# B&R Automation Studio project Nitto (part 9)

### RCP_glob.var - Package variables
```iecst
(********************************************************************
 * COPYRIGHT -- Bernecker + Rainer
 ********************************************************************
 * File: RCP_glob.var
 * Author: beutert
 * Created: September 07, 2012
 ********************************************************************
 * Global variables of project csv_bsp
 ********************************************************************)
(*======================================================================================================================================*)
(*Global recipe constants*)
(*======================================================================================================================================*)
VAR CONSTANT
	RCP_PROG_TEXT_DESCRIPTION_MAX : UINT := 79; (*maximale Anzahl von Zeichen für Beschreibungen für Rezept und Zeile*)
	RCP_PROG_TEXT_FILENAME_MAX : UINT := 29; (*maximale Anzahl von Zeichen für den Rezeptnamen*)
END_VAR
(*======================================================================================================================================*)
(*Global recipe variables*)
(*======================================================================================================================================*)
VAR
	Button : Button_typ := (0);
	ToolEdit : rcp_tool_typ := (0);
	RecipeEdit : rcp_prog_typ := (0);
	RecipeWork : rcp_prog_typ := (0);
END_VAR
```

### Glob_IO.typ - Package data types
```iecst
(********************************************************************
 * COPYRIGHT -- Bernecker + Rainer
 ********************************************************************
 * File: Glob_IO.typ
 * Author: schoenefeldr
 * Created: July 10, 2012
 ********************************************************************
 * Global data types of project 120706_hp_001
 ********************************************************************)

TYPE
	MachineIoDi_Type : 	STRUCT
		FuseFanUnwind : DiDo_Type; (*Sicherung Lüfter Abwicklung*)
		FusePlug1 : DiDo_Type; (*Sicherung OK Schukosteckdose 1*)
		FusePlug2 : DiDo_Type; (*Sicherung OK Schukosteckdose 2*)
		FusePlugCEE : DiDo_Type; (*Sicherung OK CEE-Steckdose*)
		FuseBTS : DiDo_Type; (*Sicherung OK Bahnkantensteuerung*)
		FuseQW258_262 : DiDo_Type; (*Sicherung OK QW258 - QW262*)
		FuseQW264_268 : DiDo_Type; (*Sicherung OK QW264 - QW268*)
		FuseBookletFeeder : DiDo_Type; (*Sicherung OK Booklet Feeder*)
		FuseHydraulicPump : DiDo_Type; (*Sicherung OK Hydraulikpumpe*)
		HighVoltageGenerator : DiDo_Type; (*Hochspannungsgenerator Anti-Statik OK / Ein-Aus*)
		BST_OK : DiDo_Type; (*BST OK*)
		RFK_EmcyStop_undelayed : DiDo_Type; (*RFK Not - Halt - Schütze unverzögert*)
		RFK_EmcyStop_delayed : DiDo_Type; (*RFK Not - Halt - Schütze verzögert*)
		LDT_Reset : DiDo_Type; (*LDT Reset / Steuerung Ein*)
		LDT_CtrlOff : DiDo_Type; (*LDT Steuerung Aus*)
		LDT_AutoStart_End : DiDo_Type; (*LDT Automatik Start Maschinenende*)
		LDT_AutoStart_Middle : DiDo_Type; (*LDT Automatik Start Maschinenmitte*)
		LDT_AutoStart_Unwind : DiDo_Type; (*LDT Automatik Start am Abwickler*)
		LDT_AutoStart : DiDo_Type; (*LDT Automatik Start*)
		LDT_AutoStop : DiDo_Type; (*LDT Automatik Stopp*)
		LDT_AutoStop_End : DiDo_Type; (*LDT Automatik Stopp Maschinenende*)
		LDT_AutoStop_Middle : DiDo_Type; (*LDT Automatik Stopp Maschinenmitte*)
		LDT_AutoStop_Unwind : DiDo_Type; (*LDT Automatik Stopp am Abwickler*)
		LDT_Reserve2 : DiDo_Type;
		LDT_Jog_Machine : DiDo_Type; (*LDT Jog-Mode*)
		LDT_Jog_Machine_End : DiDo_Type; (*LDT Jog-Mode Maschinenende*)
		LDT_Jog_Machine_Middle : DiDo_Type; (*LDT Jog-Mode Maschinenmitte*)
		LDT_Jog_Machine_Unwind : DiDo_Type; (*LDT Jog-Mode am Abwickler*)
		LDT_Reserve1 : DiDo_Type;
		LDT_FaultReset : DiDo_Type; (*LDT Störung quittieren*)
		LDT_UnwindMoveUp : DiDo_Type; (*LDT Abwickler heben*)
		LDT_Laminator_UpDn : DiDo_Type;
		LDT_LabelDisp_UpDn : DiDo_Type;
		LDT_UnwindMoveDown : DiDo_Type; (*LDT Abwickler senken*)
		LDT_PBS2_upDn : DiDo_Type; (*LDT Zugeinheit heben / senken*)
		LDT_LongCUTsetKnife : DiDo_Type; (*Taster zum Einsetzen der Messer*)
		LDT_PBU_upDn : DiDo_Type; (*LDT Zugstation 3 heben / senken*)
		LDT_CutTabInfeed : DiDo_Type; (*LDT Schneidetisch heben / senken Einlaufseite*)
		LDT_CutTabOutfeed : DiDo_Type; (*LDT Schneidetisch heben / senken Auslaufseite*)
		LDT_PBS1_upDn : DiDo_Type; (*LDT Zugstation 1 heben / senken*)
		LDT_LongCutUpDn : DiDo_Type; (*LDT Längsschneider heben / senken*)
		RD_UnwindTopPos : DiDo_Type; (*RD Abwickler oben*)
		RD_UnwindBotPos : DiDo_Type; (*RD Abwickler unten*)
		RD_PBS1_topPos : DiDo_Type; (*RD Zugstation 1 oben*)
		RD_PBS1_botPos : DiDo_Type; (*RD Zugstation 1 unten*)
		RD_PBU_topPos : DiDo_Type; (*RD Zugstation 3 oben*)
		RD_PBU_botPos : DiDo_Type; (*RD Zugstation 3 unten*)
		Cut1_Ref : DiDo_Type; (*Stanze 1 Referenzpunkt*)
		Cut2_Ref : DiDo_Type; (*Stanze 2 Referenzpunkt*)
		Cut3_Ref : DiDo_Type; (*Stanze 2 Referenzpunkt*)
		RD_PBS2_topPos : DiDo_Type; (*RD Zugeinheit oben*)
		RD_PBS2_botPos : DiDo_Type; (*RD Zugeinheit unten*)
		RD_LongCutTopPos : DiDo_Type; (*RD Längsschneider oben*)
		RD_LongCutBotPos : DiDo_Type; (*RD Längsschneider unten*)
		PressureCtrl : DiDo_Type; (*Druckwächter*)
		SafetyDoorInfeedCut1 : DiDo_Type; (*Safety Door Stanze 1 Infeed*)
		SafetyDoorOutfeedCut1 : DiDo_Type; (*Safety Door Stanze 1 Outfeed*)
		SafetyDoorInfeedCut2 : DiDo_Type; (*Safety Door Stanze 2 Infeed*)
		SafetyDoorOutfeedCut2 : DiDo_Type; (*Safety Door Stanze 2 Outfeed*)
		SafetyDoorInfeedCut3 : DiDo_Type; (*Safety Door Stanze 3 Infeed*)
		SafetyDoorOutfeedCut3 : DiDo_Type; (*Safety Door Stanze 3 Outfeed*)
		SafetyDoorLongCut : DiDo_Type; (*Safety Door Long cut unit*)
		SafetyDoorBooklet : DiDo_Type; (*Safety Door Long cut unit*)
		EmergencyStopCabinet : DiDo_Type; (*Not-Aus-Schalter am Schaltschrank*)
		EmergencyStopPanel : DiDo_Type; (*Not-Aus-Schalter am Panel*)
		EmergencyStopUnwinder : DiDo_Type; (*Not-Aus-Schalter am Abwickler*)
		EmergencyStopBooklet : DiDo_Type; (*Not-Aus-Schalter am Schaltschrank*)
		EmergencyStopLongCut : DiDo_Type; (*Not-Aus-Schalter am Längsschneider*)
		EmergencyStopPullWire : DiDo_Type; (*Not-Aus-Schalter am Längsschneider*)
		LightSensorConvBelt : DiDo_Type; (*Lichttaster Auslageband*)
		EmergencyStopTandemWinder : DiDo_Type; (*Not-Aus-Schalter am Tandemwickler*)
		EmergencyStopEndModule : DiDo_Type; (*Not-Aus-Schalter am Ende der Maschine*)
		EmergencyStopMiddle : DiDo_Type; (*Not-Aus-Schalter in der Mitte der Maschine*)
		RD_LaminatorTopPos : DiDo_Type;
		RD_LaminatorBotPos : DiDo_Type;
		LT_LabelDisp_LoopUnwinder : DiDo_Type;
		LT_LabelDisp_LoopWinder : DiDo_Type;
		LT_LabelDisp_WebBreak1 : DiDo_Type;
		LT_LabelDisp_WebBreak2 : DiDo_Type;
		LabelDisp_RegMark1 : DiDo_Type;
		LabelDisp_RegMark2 : DiDo_Type;
		Fuse_Laminator1 : DiDo_Type;
		Fuse_Laminator2 : DiDo_Type;
		Fuse_GridWinder1 : DiDo_Type;
		Fuse_LabelDisp1 : DiDo_Type;
		Fuse_LabelDisp2 : DiDo_Type;
		TopWindSpikeSuppClosed : DiDo_Type;
		Liner_detekce : DiDo_Type;
		BotWindSpikeSuppClosed : DiDo_Type;
	END_STRUCT;
	MachineIo_Type : 	STRUCT
		DIn : MachineIoDi_Type;
		DOut : MachineIoDo_Type;
		AIn : MachineIoAi_Type;
		AOut : MachineIoAo_Type;
	END_STRUCT;
	MachineIoDo_Type : 	STRUCT
		CtrlPowerEmcyUndel : DiDo_Type; (*24V DC Versorgung nach Not-Halt*)
		CtrlPowerEmcyDel : DiDo_Type; (*24V DC Versorgung nach Not-Halt zeitverzögert*)
		EnabDrives : DiDo_Type; (*Enable ACOPOS-Multi*)
		ContactSuction : DiDo_Type; (*potentialfreier Kontakt Absaugung Ein*)
		Plug1_OnOff : DiDo_Type; (*Schukosteckdose 1 Ein / Aus*)
		Plug2_OnOff : DiDo_Type; (*Schukosteckdose 2 Ein / Aus*)
		PlugCEE_OnOff : DiDo_Type; (*CEE-Steckdose 16A Ein / Aus*)
		HydraulicPumpOn : DiDo_Type; (*Schütz Hydraulikpumpe ein*)
		BST_Enable : DiDo_Type; (*BST Freigabe*)
		BST_Manual : DiDo_Type; (*BST Handbetrieb*)
		BST_Neutral : DiDo_Type; (*BST Mittenstellung*)
		BST_Automatic : DiDo_Type; (*BST Mittenstellung*)
		BST_ArrowLeft : DiDo_Type; (*BST Pfeil links BST Tastatursperre*)
		BST_ArrowRight : DiDo_Type; (*BST Pfeil rechts BST Tastatursperre*)
		LampGreen : DiDo_Type; (*Turmleuchte grün*)
		LampYellow : DiDo_Type; (*Turmleuchte gelb*)
		LampRed : DiDo_Type; (*Turmleuchte rot*)
		TowerHorn : DiDo_Type; (*Turmleuchte Hupe*)
		VentLabelDisp : DiDo_Type; (*Ventil Label Dispenser Up Down*)
		VentLaminatorMoveUp : DiDo_Type; (*Ventil Abwickler heben*)
		VentLaminatorMoveDown : DiDo_Type; (*Ventil Abwickler heben*)
		VentUnwindMoveUp : DiDo_Type; (*Ventil Laminierer heben*)
		VentUnwindMoveDown : DiDo_Type; (*Ventil Laminierer senken*)
		VentCutTabInfeedMoveUpDn : DiDo_Type; (*Ventil Schneidetisch heben / senken Einlaufseite*)
		VentCutTabOutfeedMoveUpDn : DiDo_Type; (*Ventil Schneidetisch heben / senken Auslaufseite*)
		Vent1Dancer : DiDo_Type; (*Ventil 1 Tänzer*)
		VentAirSupply : DiDo_Type; (*Hauptventil*)
		VentPBS1_MoveDown : DiDo_Type; (*Ventil Zugstation 1 senken*)
		VentPBS1_MoveUp : DiDo_Type; (*Ventil Zugstation 1 heben*)
		VentPBU_MoveUP : DiDo_Type; (*Ventil Zugstation 3 heben*)
		VentPBU_MoveDown : DiDo_Type; (*Ventil Zugstation 3 senken*)
		VentPBS2_MoveDown : DiDo_Type; (*Ventil Zugeinheit senken*)
		VentLongCutMoveUp : DiDo_Type; (*Ventil Längsschneider heben*)
		VentLongCutSetKnifeIn : DiDo_Type; (*Ventil Längsschneider Messer setzen*)
		VentLongCutSetKnifeOut : DiDo_Type; (*Ventil Längsschneider Messer setzen*)
		VentLongCutMoveDown : DiDo_Type; (*Ventil Längsschneider senken *)
		ValveCuttingUnitToolUp : DiDo_Type; (*Ventil Stanzstation Werkzeug heben*)
		ValveCut1BridgeDown : DiDo_Type; (*Ventil Stanzstation1 Brücke senken*)
		ValveCut2BridgeDown : DiDo_Type; (*Ventil Stanzstation 2 Brücke senken*)
		ValveCut3BridgeDown : DiDo_Type; (*Ventil Stanzstation 3 Brücke senken*)
		BookletFeederREG : DiDo_Type; (*Ventil Stanzstation 3 Brücke senken*)
		BookletFeederON : DiDo_Type; (*Ventil Stanzstation 3 Brücke senken*)
	END_STRUCT;
	MachineIoAo_Type : 	STRUCT
		MagBrakeUnwind : AiAo_Type; (*Ansteuerung Magnetpulverbremse Abwickler*)
		VentDancer : AiAo_Type; (*Proportionalventil Tänzerspannung (Festo)*)
		VentClutchSpend1 : AiAo_Type; (*Proportionalventil Rutschkupplung Abwickler 1*)
		VentClutchSpend2 : AiAo_Type; (*Proportionalventil Rutschkupplung Abwickler 2*)
		VentClutchSpend3 : AiAo_Type; (*Proportionalventil Rutschkupplung Abwickler 3*)
		VentClutchLaminator1 : AiAo_Type; (*Proportionalventil Rutschkupplung Abwickler 3*)
		VentClutchLaminator2 : AiAo_Type; (*Proportionalventil Rutschkupplung Abwickler 3*)
		VentClutchGrid1 : AiAo_Type; (*Proportionalventil Rutschkupplung Gitteraufwickler 1*)
		VentClutchGrid2 : AiAo_Type; (*Proportionalventil Rutschkupplung Gitteraufwickler 2*)
		VentOptClutchTUnwindTop : AiAo_Type; (*Option Proportionalventil Rutschkupplung Tandemwickler oben*)
		VentOptClutchTUnwindBot : AiAo_Type; (*Option Proportionalventil Rutschkupplung Tandemwickler unten*)
	END_STRUCT;
	MachineIoAi_Type : 	STRUCT
		FlengeDMS : AiAo_Type; (*Flanschkraftaufnehmer*)
		FDriveSideCut1 : AiAo_Type; (*Stanze 1 Druckkraftaufnehmer Antriebsseite*)
		FOperatorSideCut1 : AiAo_Type; (*Stanze 1 Druckkraftaufnehmer Bedienerseite*)
		FDriveSideCut2 : AiAo_Type; (*Stanze 2 Druckkraftaufnehmer Antriebsseite*)
		FOperatorSideCut2 : AiAo_Type; (*Stanze 2 Druckkraftaufnehmer Bedienerseite*)
		FDriveSideCut3 : AiAo_Type; (*Stanze 3 Druckkraftaufnehmer Antriebsseite*)
		FOperatorSideCut3 : AiAo_Type; (*Stanze 3 Druckkraftaufnehmer Bedienerseite*)
		DiamMainUnwind : AiAo_Type; (*Durchmesserabfrage Abwicklung*)
		DiamSpend1 : AiAo_Type; (*Durchmesserabfrage Abwickler 1*)
		DiamSpend2 : AiAo_Type; (*Durchmesserabfrage Abwickler 2*)
		DiamLaminator1 : AiAo_Type; (*Durchmesserabfrage Laminierer 1*)
		DiamLaminator2 : AiAo_Type; (*Durchmesserabfrage Laminierer 2*)
		DiamGrid1 : AiAo_Type; (*Durchmesserabfrage Gitteraufwickler 1*)
		DiamGrid2 : AiAo_Type; (*Durchmesserabfrage Gitteraufwickler 2*)
		DancerPos : AiAo_Type; (*Tänzerlage*)
		DiamTUnwindTop : AiAo_Type; (*Durchmesserabfrage Tandemwickler oben*)
		DiamTUnwindBot : AiAo_Type; (*Durchmesserabfrage Tandemwickler unten*)
		Dancer_position : AiAo_Type; (*pozice danceru optický senzor*)
		TestSensor : AiAo_Type; (*Durchmesserabfrage Tandemwickler unten*)
	END_STRUCT;
END_TYPE
```

### Library Logical/Bibliothek (IEC) - Eine neue Quellbibliothek

#### Package Logical/Bibliothek/CONST - Neues leeres Paket

#### FB_CONST_AXISSTATE.st
```iecst
(********************************************************************
 * COPYRIGHT -- Microsoft
 ********************************************************************
 * Library: Bibliothek
 * Datei: FB_CONST_AXISSTATE.st
 * Autor: awalz
 * Erstellt: 26. August 2014
 ********************************************************************
 * Implementierung der Library Bibliothek
 ********************************************************************)

(* TODO: Bitte Kommentar hier einfügen *)
FUNCTION_BLOCK FB_CONST_AXIS_STATE
END_FUNCTION_BLOCK
```

#### FB_CONST_UNIT_MODES.st
```iecst
(********************************************************************
 * COPYRIGHT -- Microsoft
 ********************************************************************
 * Library: Bibliothek
 * Datei: FB_CONST_UNIT_MODES.st
 * Autor: Awalz
 * Erstellt: 7. Mai 2014
 ********************************************************************
 * Implementierung der Library Bibliothek
 ********************************************************************)

 (*<$Description$> TODO: Bitte Kommentar hier einzufügen </$Description$>*)
FUNCTION_BLOCK FB_CONST_UNIT_MODES
END_FUNCTION_BLOCK
```

#### FB_CONST_CUTTINGUNIT_CMDS.st
```iecst
(********************************************************************
 * COPYRIGHT -- Microsoft
 ********************************************************************
 * Library: Bibliothek
 * Datei: FB_CONST_CUTTINGUNIT_CMDS.st
 * Autor: Awalz
 * Erstellt: 7. Mai 2014
 ********************************************************************
 * Implementierung der Library Bibliothek
 ********************************************************************)

 (*<$Description$> TODO: Bitte Kommentar hier einzufügen </$Description$>*)
FUNCTION_BLOCK FB_CONST_CUTTINGUNIT_CMDS
END_FUNCTION_BLOCK
```

#### FB_CONST_CUTTINGUNIT_MODES.st
```iecst
(********************************************************************
 * COPYRIGHT -- Microsoft
 ********************************************************************
 * Library: Bibliothek
 * Datei: FB_CONST_CUTTINGUNIT_MODES.st
 * Autor: Awalz
 * Erstellt: 7. Mai 2014
 ********************************************************************
 * Implementierung der Library Bibliothek
 ********************************************************************)

 (*<$Description$> TODO: Bitte Kommentar hier einzufügen </$Description$>*)
FUNCTION_BLOCK FB_CONST_CUTTINGUNIT_MODES
END_FUNCTION_BLOCK
```

#### FB_CONST_MASCHINE.st
```iecst
(********************************************************************
 * COPYRIGHT -- Microsoft
 ********************************************************************
 * Library: Bibliothek
 * Datei: FB_CONST_MASCHINE.st
 * Autor: Awalz
 * Erstellt: 1. April 2014
 ********************************************************************
 * Implementierung der Library Bibliothek
 ********************************************************************)

 (*<$Description$> TODO: Bitte Kommentar hier einzufügen </$Description$>*)
FUNCTION_BLOCK FB_CONST_MASCHINE
END_FUNCTION_BLOCK
```

#### FB_CONST_AXIS_ACTIONS.st
```iecst
(********************************************************************
 * COPYRIGHT -- Microsoft
 ********************************************************************
 * Library: Bibliothek
 * Datei: FB_CONST_AXIS_ACTIONS.st
 * Autor: Awalz
 * Erstellt: 1. April 2014
 ********************************************************************
 * Implementierung der Library Bibliothek
 ********************************************************************)

 (*<$Description$> TODO: Bitte Kommentar hier einzufügen </$Description$>*)
FUNCTION_BLOCK FB_CONST_AXIS_ACTIONS
END_FUNCTION_BLOCK
```

#### FB_CONST_MACHINE_MODE.st
```iecst
(********************************************************************
 * COPYRIGHT -- Microsoft
 ********************************************************************
 * Library: Bibliothek
 * Datei: FB_CONST_MACHINE_MODE.st
 * Autor: Awalz
 * Erstellt: 31. März 2014
 ********************************************************************
 * Implementierung der Library Bibliothek
 ********************************************************************)

 (*<$Description$> TODO: Bitte Kommentar hier einzufügen </$Description$>*)
FUNCTION_BLOCK FB_CONST_MACHINE_MODES
END_FUNCTION_BLOCK
```

#### FB_CONST_LAMP.st
```iecst
(********************************************************************
 * COPYRIGHT -- Microsoft
 ********************************************************************
 * Library: Bibliothek
 * Datei: FB_CONST_LAMP.st
 * Autor: Awalz
 * Erstellt: 30. April 2014
 ********************************************************************
 * Implementierung der Library Bibliothek
 ********************************************************************)

 (*<$Description$> TODO: Bitte Kommentar hier einzufügen </$Description$>*)
FUNCTION_BLOCK FB_CONST_LAMP
END_FUNCTION_BLOCK
```

#### FB_CONST_CUTTINGUNIT.st
```iecst
(********************************************************************
 * COPYRIGHT -- Microsoft
 ********************************************************************
 * Library: Bibliothek
 * Datei: FB_CONST_CUTTINGUNIT.st
 * Autor: Awalz
 * Erstellt: 7. Mai 2014
 ********************************************************************
 * Implementierung der Library Bibliothek
 ********************************************************************)

 (*<$Description$> TODO: Bitte Kommentar hier einzufügen </$Description$>*)
FUNCTION_BLOCK FB_CONST_CUTTINGUNIT
END_FUNCTION_BLOCK
```

#### FB_CUTTINGUNIT_CMD.st
```iecst
(********************************************************************
 * COPYRIGHT -- Microsoft
 ********************************************************************
 * Library: Bibliothek
 * Datei: FB_CUTTINGUNIT_CMD.st
 * Autor: Awalz
 * Erstellt: 7. Mai 2014
 ********************************************************************
 * Implementierung der Library Bibliothek
 ********************************************************************)

 (*<$Description$> TODO: Bitte Kommentar hier einzufügen </$Description$>*)
FUNCTION_BLOCK FB_CUTTINGUNIT_CMD
	IF set THEN
		IF value < CONST.CUTTINGUNIT.CMDs.NO_CMD OR value > CONST.CUTTINGUNIT.CMDs.ABORT THEN
			text := '******';
		ELSE
			text := CONST.CUTTINGUNIT.CMDs.texts[value];
		END_IF
	END_IF
END_FUNCTION_BLOCK
```

#### FB_CUTTING_MODE.st
```iecst
(********************************************************************
 * COPYRIGHT -- Microsoft
 ********************************************************************
 * Library: Bibliothek
 * Datei: FB_CUTTING_MODE.st
 * Autor: Awalz
 * Erstellt: 20. Mai 2014
 ********************************************************************
 * Implementierung der Library Bibliothek
 ********************************************************************)

 (*<$Description$> TODO: Bitte Kommentar hier einzufügen </$Description$>*)
FUNCTION_BLOCK FB_CUTTING_MODE
END_FUNCTION_BLOCK
```

#### FB_CONST_CUTTINGUNIT_TOOLS.st
```iecst
(********************************************************************
 * COPYRIGHT -- Microsoft
 ********************************************************************
 * Library: Bibliothek
 * Datei: FB_CONST_CUTTINGUNIT_TOOLS.st
 * Autor: okrebs
 * Erstellt: 23. Mai 2014
 ********************************************************************
 * Implementierung der Library Bibliothek
 ********************************************************************)

(* TODO: Bitte Kommentar hier einzufügen *)
FUNCTION_BLOCK FB_CONST_CUTTINGUNIT_TOOLS
END_FUNCTION_BLOCK
```

#### FB_CONST_ALARMS.st
```iecst
(********************************************************************
 * COPYRIGHT -- Microsoft
 ********************************************************************
 * Library: Bibliothek
 * Datei: FB_CONST_ALARMS.st
 * Autor: awalz
 * Erstellt: 1. August 2014
 ********************************************************************
 * Implementierung der Library Bibliothek
 ********************************************************************)

(* TODO: Bitte Kommentar hier einfügen *)
FUNCTION_BLOCK FB_CONST_ALARMS
END_FUNCTION_BLOCK
```

#### FB_CONST_CUTTINGUNIT_ERRORS.st
```iecst
(********************************************************************
 * COPYRIGHT -- Microsoft
 ********************************************************************
 * Library: Bibliothek
 * Datei: FB_CONST_CUTTINGUNIT_ERRORS.st
 * Autor: okrebs
 * Erstellt: 23. Mai 2014
 ********************************************************************
 * Implementierung der Library Bibliothek
 ********************************************************************)

(* TODO: Bitte Kommentar hier einzufügen *)
FUNCTION_BLOCK FB_CONST_CUTTINGUNIT_ERRORS
END_FUNCTION_BLOCK
```

#### Package Logical/Bibliothek/Genarals - Neues leeres Paket

#### FB_Lamp.st
```iecst
(********************************************************************
 * COPYRIGHT -- Microsoft
 ********************************************************************
 * Library: Bibliothek
 * Datei: FB_Lamp.st
 * Autor: Awalz
 * Erstellt: 12. Mai 2014
 ********************************************************************
 * Implementierung der Library Bibliothek
 ********************************************************************)

 (*<$Description$> TODO: Bitte Kommentar hier einzufügen </$Description$>*)
FUNCTION_BLOCK FB_Lamp
 rtrig(CLK := button);
	ftrig(CLK := button);
 	IF aktion = CONST.LAMP.OFF THEN
 		output := FALSE;
	ELSIF aktion = CONST.LAMP.ON THEN
		output := TRUE;
	ELSIF aktion = CONST.LAMP.BLINK200 THEN
		output := clk.c200.Output;
	ELSIF aktion = CONST.LAMP.BLINK500 THEN
		output := clk.c500.Output;
	ELSIF aktion = CONST.LAMP.BLINK1000 THEN
		output := clk.c1000.Output;
	ELSIF aktion = CONST.LAMP.BLINK5000 THEN
		output := clk.c5000.Output;
	END_IF

	led := output;
	ledinv := NOT output;

END_FUNCTION_BLOCK
```

#### FB_Clk.st
```iecst
(********************************************************************
 * COPYRIGHT -- Microsoft
 ********************************************************************
 * Library: Bibliothek
 * Datei: FB_Clk.st
 * Autor: Awalz
 * Erstellt: 30. April 2014
 ********************************************************************
 * Implementierung der Library Bibliothek
 ********************************************************************)

 (*<$Description$> TODO: Bitte Kommentar hier einzufügen </$Description$>*)
FUNCTION_BLOCK FB_Clk
	c200();
	c500();
	c1000();
	c5000();
END_FUNCTION_BLOCK
```

#### FB_KeyLamp.st
```iecst
(********************************************************************
 * COPYRIGHT -- Microsoft
 ********************************************************************
 * Library: Bibliothek
 * Datei: FB_KeyLamp.st
 * Autor: Awalz
 * Erstellt: 12. Mai 2014
 ********************************************************************
 * Implementierung der Library Bibliothek
 ********************************************************************)

 (*<$Description$> TODO: Bitte Kommentar hier einzufügen </$Description$>*)
FUNCTION_BLOCK FB_KeyLamp
		LDT( clk := clk );
END_FUNCTION_BLOCK
```

#### FB_Ampel.st
```iecst
(********************************************************************
 * COPYRIGHT -- Microsoft
 ********************************************************************
 * Library: Bibliothek
 * Datei: FB_Ampel.st
 * Autor: Awalz
 * Erstellt: 12. Mai 2014
 ********************************************************************
 * Implementierung der Library Bibliothek
 ********************************************************************)

 (*<$Description$> TODO: Bitte Kommentar hier einzufügen </$Description$>*)
FUNCTION_BLOCK FB_Ampel
	rtrig(CLK := horn);
	hornPuls(clk := clk);
	Rot(clk := clk);
	Gelb(clk := clk);
	Gruen(clk := clk);
	timer_TOF(IN := rtrig.Q, PT := ondelay);
//	horn_o := timer_TOF.Q;
	horn_o := SEL (timer_TOF.Q, hornPuls.led, timer_TOF.Q); (* pulsierendes Hupen zu erzeugen das Signal wird durch hornPuls von Aussen getaktet*)
END_FUNCTION_BLOCK
```

#### FB_ModulStatus.st
```iecst
(********************************************************************
 * COPYRIGHT -- Microsoft
 ********************************************************************
 * Library: Bibliothek
 * Datei: FB_ModulStatus.st
 * Autor: Awalz
 * Erstellt: 12. Mai 2014
 ********************************************************************
 * Implementierung der Library Bibliothek
 ********************************************************************)

 (*<$Description$> TODO: Bitte Kommentar hier einzufügen </$Description$>*)
FUNCTION_BLOCK FB_ModulStatus
	IF axisState.ContinuousMotion THEN
		AxisState_status := 'ContinuousMotion';
	ELSIF axisState.Disabled THEN
		AxisState_status := 'Disabled';
	ELSIF axisState.DiscreteMotion THEN
		AxisState_status := 'DiscreteMotion';
	ELSIF axisState.Error THEN
		AxisState_status := 'Error';
	ELSIF axisState.Errorstop THEN
		AxisState_status := 'Errorstop';
	ELSIF axisState.StandStill THEN
		AxisState_status := 'StandStill';
	ELSIF axisState.Stopping THEN
		AxisState_status := 'Stopping';
	ELSIF axisState.SynchronizedMotion THEN
		AxisState_status := 'SynchronizedMotion';
	END_IF
END_FUNCTION_BLOCK
```

#### FB_UnitChkStatus.st
```iecst
(********************************************************************
 * COPYRIGHT -- Microsoft
 ********************************************************************
 * Library: Bibliothek
 * Datei: FB_UnitChkStatus.st
 * Autor: Awalz
 * Erstellt: 12. Mai 2014
 ********************************************************************
 * Implementierung der Library Bibliothek
 ********************************************************************)

 (*<$Description$> TODO: Bitte Kommentar hier einzufügen </$Description$>*)
FUNCTION_BLOCK FB_UnitChkStatus
	IF enable THEN
		IF setMode = status.mode THEN
			IF setMode = CONST.UNITMODEs.DISABLE THEN
				ready := NOT status.isCoupled;
			ELSIF setMode = CONST.UNITMODEs.ENABLE THEN
				ready := status.isCoupled;
			ELSE
				ready := FALSE;
			END_IF
		ELSE
			ready := FALSE;
		END_IF
	END_IF

	status.ready := ready;
END_FUNCTION_BLOCK
```

#### FB_ClkPulse.st
```iecst
(********************************************************************
 * COPYRIGHT -- Microsoft
 ********************************************************************
 * Library: Bibliothek
 * Datei: FB_ClkPulse.st
 * Autor: Awalz
 * Erstellt: 30. April 2014
 ********************************************************************
 * Implementierung der Library Bibliothek
 ********************************************************************)

 (*<$Description$> TODO: Bitte Kommentar hier einzufügen </$Description$>*)
FUNCTION_BLOCK FB_ClkPulse

CASE state OF
	CLOCK_ON:
		IF enable THEN
			Output := TRUE;
			timer(IN := FALSE);
			timer(IN := TRUE, PT := TimeOn);
		  	state:= CLOCK_WAIT_ON;
		END_IF

	CLOCK_WAIT_ON:
		timer();
		IF NOT enable THEN
			timer(IN := FALSE);
			Output := FALSE;
			state := CLOCK_ON;
		ELSIF timer.Q THEN
			timer(IN := FALSE);
			Output := FALSE;
			timer(IN := TRUE, PT := TimeOff);
	   		state := CLOCK_WAIT_OFF;
		END_IF

	CLOCK_WAIT_OFF:
		timer();
		IF NOT enable THEN
			timer(IN := FALSE);
			Output := FALSE;
			state := CLOCK_ON;
		ELSIF timer.Q THEN
			Output := TRUE;
			timer(IN := FALSE);
			timer(IN := TRUE, PT := TimeOn);
		   	state:= CLOCK_WAIT_ON;
		END_IF
	ELSE  						(* Unknown program state *)
		state:= CLOCK_ON;
	END_CASE
END_FUNCTION_BLOCK
```

#### FB_ErrorHdl.st
```iecst
(********************************************************************
 * COPYRIGHT -- Microsoft
 ********************************************************************
 * Library: Bibliothek
 * Datei: FB_ErrorHdl.st
 * Autor: Awalz
 * Erstellt: 12. Mai 2014
 ********************************************************************
 * Implementierung der Library Bibliothek
 ********************************************************************)

 (*<$Description$> TODO: Bitte Kommentar hier einzufügen </$Description$>*)
FUNCTION_BLOCK FB_ErrorHdl
	IF reset THEN
		id := 0;
		state := 0;
		text :='';
		fnc :='';
		flag := FALSE;
		reset := FALSE;
	END_IF
	IF set THEN
		flag := TRUE;
		set := FALSE;
	END_IF
END_FUNCTION_BLOCK
```

#### FB_Panel.st
```iecst
(********************************************************************
 * COPYRIGHT -- Microsoft
 ********************************************************************
 * Library: Bibliothek
 * Datei: FB_Panel.st
 * Autor: Awalz
 * Erstellt: 12. Mai 2014
 ********************************************************************
 * Implementierung der Library Bibliothek
 ********************************************************************)

 (*<$Description$> TODO: Bitte Kommentar hier einzufügen </$Description$>*)
FUNCTION_BLOCK FB_Panel
		clk();
		Emergency (clk := clk);

		EMCY_Button_o.0 := EMCY_Button;
		LDTRESET(clk := clk);
		LDTStop (clk := clk);
		LDTAutomatic (clk := clk);
		LDTControlON(clk := clk);
		LDTControlOFF(clk := clk);
		LDTJOG(clk := clk);
END_FUNCTION_BLOCK
```

#### FB_PullBreakClampToggle.st
```iecst
(********************************************************************
 * COPYRIGHT -- Microsoft
 ********************************************************************
 * Library: Bibliothek
 * Datei: FB_PullBreakClampToggle.st
 * Autor: Awalz
 * Erstellt: 12. Mai 2014
 ********************************************************************
 * Implementierung der Library Bibliothek
 ********************************************************************)

 (*<$Description$> TODO: Bitte Kommentar hier einzufügen </$Description$>*)
FUNCTION_BLOCK FB_PullBreakClampToggle
buttomToggle(clk := clk);
	IF enable THEN
		IF buttomToggle.LDT.rtrig.Q (*AND NOT buttomToggle2.LDT.rtrig.Q *)THEN
			IF NOT onewayini THEN
				IF isup THEN (*Sensorausgang *)
					toUp_o := FALSE;
					toDown_o := TRUE;
				ELSE
					toDown_o := FALSE;
					toUp_o := TRUE;
				END_IF
		 	ELSE
		 		IF isdown THEN
					toDown_o := FALSE;
					toUp_o := TRUE;
				ELSE
					toDown_o :=TRUE;
					toUp_o := FALSE;
				END_IF
			END_IF
		END_IF

			IF isdown AND buttomToggle2.LDT.button AND (state = 0) THEN
				limiterForward_o := FALSE;
				limiterBackward_o := TRUE;
				Time1.IN := TRUE;
				Time1.PT := T#3s;
				state := 1;
			ELSIF buttomToggle2.LDT.button AND (state = 0) THEN
				limiterForward_o := TRUE;
				limiterBackward_o := FALSE;
				toDown_o := TRUE;
				toUp_o := FALSE;
				state := 0;
			END_IF
			IF NOT limiterSwitchDrvSide AND NOT limiterSwitchOpSide AND Time1.Q AND (state = 1) THEN
				Time1.IN := FALSE;
				toDown_o := FALSE;
				toUp_o := TRUE;
				state := 0;
			END_IF

			Time1();
	ELSE
//		toDown_o :=FALSE;
//		toUp_o := FALSE;
	END_IF
	IF init THEN
		toUp_o := TRUE;
		init := FALSE;
	END_IF

	IF 	 NOT onewayini THEN
		buttomToggle.LDT.aktion := SEL((toUp_o AND isup), CONST.LAMP.OFF, CONST.LAMP.ON);
	ELSE
		buttomToggle.LDT.aktion := SEL((toUp_o AND NOT isdown ), CONST.LAMP.OFF, CONST.LAMP.ON);
	END_IF

END_FUNCTION_BLOCK
```

#### FB_Safety.st
```iecst
(********************************************************************
 * COPYRIGHT -- Microsoft
 ********************************************************************
 * Library: Bibliothek
 * Datei: FB_Safety.st
 * Autor: Awalz
 * Erstellt: 12. Mai 2014
 ********************************************************************
 * Implementierung der Library Bibliothek
 ********************************************************************)

 (*<$Description$> TODO: Bitte Kommentar hier einzufügen </$Description$>*)
FUNCTION_BLOCK FB_Safety
END_FUNCTION_BLOCK
```

#### FB_PowerBridge.st
```iecst
(********************************************************************
 * COPYRIGHT -- Microsoft
 ********************************************************************
 * Library: Bibliothek
 * Datei: FB_PowerBridge.st
 * Autor: Awalz
 * Erstellt: 2. Juni 2014
 ********************************************************************
 * Implementierung der Library Bibliothek
 ********************************************************************)

 (*<$Description$> TODO: Bitte Kommentar hier einzufügen </$Description$>*)
FUNCTION_BLOCK FB_PowerBridge
	toggle(clk:= clk);
	movebutton(clk := clk);
	bridgedownbutton(clk := clk);
	KNpressureOperside := INT_TO_REAL (pressureOperside) * SCALE_10V_TO_KN;
	KNpressuredrvside  := INT_TO_REAL (pressuredrvside) * SCALE_10V_TO_KN;
	IF withpressureSensor THEN
		 IF KNpressuredrvside > pressurereference OR KNpressureOperside >  pressurereference THEN   (**)
			pressurepresent := TRUE;
		ELSE
			pressurepresent := FALSE;
		END_IF
	ELSE
		IF button THEN
			pressurepresent := TRUE;
			valveOut := TRUE;
		ELSE
			pressurepresent := FALSE;
			valveOut := FALSE;
		END_IF
	END_IF

END_FUNCTION_BLOCK
```

#### FB_MessageInstance.st
```iecst
(********************************************************************
 * COPYRIGHT -- Microsoft
 ********************************************************************
 * Library: Bibliothek
 * Datei: FB_MessageInstance.st
 * Autor: Awalz
 * Erstellt: 14. Mai 2014
 ********************************************************************
 * Implementierung der Library Bibliothek
 ********************************************************************)

 (*<$Description$> TODO: Bitte Kommentar hier einzufügen </$Description$>*)
FUNCTION_BLOCK FB_MessageInstance
END_FUNCTION_BLOCK
```

#### FB_limitswitch.st
```iecst
(********************************************************************
 * COPYRIGHT -- Microsoft
 ********************************************************************
 * Library: Bibliothek
 * Datei: FB_limitswitch.st
 * Autor: awalz
 * Erstellt: 26. Juni 2014
 ********************************************************************
 * Implementierung der Library Bibliothek
 ********************************************************************)

(* TODO: Bitte Kommentar hier einfügen *)
FUNCTION_BLOCK FB_limitswitch
END_FUNCTION_BLOCK
```

#### FB_Hydraulic.st
```iecst
(********************************************************************
 * COPYRIGHT -- Microsoft
 ********************************************************************
 * Library: Bibliothek
 * Datei: FB_Hydraulic.st
 * Autor: Awalz
 * Erstellt: 23. Juni 2014
 ********************************************************************
 * Implementierung der Library Bibliothek
 ********************************************************************)

(* TODO: Bitte Kommentar hier einfügen *)
FUNCTION_BLOCK FB_Hydraulic
IF  enable THEN
	IF buttonUp AND NOT buttonDown AND NOT limitswitch THEN
		go_up := TRUE;
		LED_is_up:= TRUE;
		LED_is_down := FALSE;
		commonValve:=TRUE;(*main Valve right or left side*)
		pumpe:=TRUE;
	ELSIF buttonDown AND NOT buttonUp THEN
		go_up := FALSE;
		LED_is_down:=TRUE;
		commonValve:=TRUE;
	ELSIF NOT buttonDown AND NOT buttonUp THEN
		go_up := FALSE;
		LED_is_down := FALSE;
		commonValve:=FALSE;
		pumpe:=FALSE;
	END_IF
	IF limitswitch THEN
		LED_is_up :=TRUE;
		pumpe :=FALSE;
	ELSE
		LED_is_up :=FALSE;
	END_IF
ELSE
	go_up := FALSE;
	commonValve:=FALSE;
	pumpe:=FALSE;
	LED_is_down := FALSE;
END_IF
END_FUNCTION_BLOCK
```

#### FB_TurnGrWinKeysbox.st
```iecst
(********************************************************************
 * COPYRIGHT -- Microsoft
 ********************************************************************
 * Library: Bibliothek
 * Datei: FB_TurnGrWinKeysbox.st
 * Autor: Awalz
 * Erstellt: 5. Juni 2014
 ********************************************************************
 * Implementierung der Library Bibliothek
 ********************************************************************)

 (*<$Description$> TODO: Bitte Kommentar hier einzufügen </$Description$>*)
FUNCTION_BLOCK FB_TurnGrWinKeysbox
		GridWinrightkey(clk := clk);   (**)
		GridWinleftkey(clk := clk);
		feederturnkey(clk := clk);
		IF feederturnkey.LDT.rtrig.Q THEN
			(*feederlimitswitch:	BOOL;*)
			feederturn:= TRUE;
		(*	feederFUright:BOOL;*)
		ELSE
			feederturn:= FALSE;
		END_IF
END_FUNCTION_BLOCK
```

#### FB_WebGuiding.st
```iecst
(********************************************************************
 * COPYRIGHT -- Microsoft
 ********************************************************************
 * Library: Bibliothek
 * Datei: FB_WebGuiding.st
 * Autor: awalz
 * Erstellt: 27. Juni 2014
 ********************************************************************
 * Implementierung der Library Bibliothek
 ********************************************************************)

(* TODO: Bitte Kommentar hier einfügen *)
FUNCTION_BLOCK FB_WebGuiding

	hardwareActive := hardwareOK; // Meldund für Visu Bahnkantenregelung ok

	IF enable THEN
		active := 1;
	ELSE
		active := 0;
	END_IF;

	handtrigg(CLK:= hand);
	centertrigg(CLK:=center);
	autotrigg(CLK := auto);
	IF centertrigg.Q(*center*) AND NOT TP_01.Q THEN
		manual := FALSE;
		neutral := TRUE;
		automatic:= FALSE;
		Start_timer := TRUE;
		centerSelect := TRUE;
		handSelect := FALSE;
		autoSelect := FALSE;

	ELSIF handtrigg.Q	(*hand*) AND NOT TP_01.Q THEN
		manual := TRUE;
		automatic:= FALSE;
		neutral := FALSE;
		centerSelect:= FALSE;
		handSelect := TRUE;
		autoSelect := FALSE;
		Start_timer := TRUE;

	ELSIF autotrigg.Q	(*auto*) AND  NOT TP_01.Q THEN
		neutral  := FALSE;
		manual := FALSE;
		automatic:= TRUE;
		Start_timer := TRUE;
		centerSelect:= FALSE;
		handSelect := FALSE;
		autoSelect := TRUE;
	ELSE

	END_IF;

	TP_01( IN:= Start_timer,PT:= T#1100ms);
	Start_timer := FALSE;
	IF NOT  TP_01.Q THEN
		neutral  := FALSE;
		manual := FALSE;
		automatic:= FALSE;

	END_IF;

	IF handSelect  THEN
		IF moveRight THEN
			arrowLeft  := TRUE;
		ELSE
			arrowLeft  := FALSE;
		END_IF;
		IF	moveLeft THEN
			arrowRight := TRUE;
		ELSE
			arrowRight:= FALSE;
		END_IF

	END_IF
END_FUNCTION_BLOCK
```

#### FB_StartStopbox.st
```iecst
(********************************************************************
 * COPYRIGHT -- Microsoft
 ********************************************************************
 * Library: Bibliothek
 * Datei: FB_StartStopbox.st
 * Autor: awalz
 * Erstellt: 27. Juni 2014
 ********************************************************************
 * Implementierung der Library Bibliothek
 ********************************************************************)

(* TODO: Bitte Kommentar hier einfügen *)
FUNCTION_BLOCK FB_StartStopbox
	start(clk:= clk);
	stop(clk := clk);
	jog(clk := clk);
	clk();
END_FUNCTION_BLOCK
```

#### FB_SummeryStarStop.st
```iecst
(********************************************************************
 * COPYRIGHT -- Microsoft
 ********************************************************************
 * Library: Bibliothek
 * Datei: FB_SummeryStarStop.st
 * Autor: awalz
 * Erstellt: 27. Juni 2014
 ********************************************************************
 * Implementierung der Library Bibliothek
 ********************************************************************)

(* TODO: Bitte Kommentar hier einfügen *)
FUNCTION_BLOCK FB_SummeryStarStop
	IF 	boxunwinder.jog.LDT.button OR boxwebbuffer.jog.LDT.button OR boxcutting1.jog.LDT.button
		OR boxlongcutter.jog.LDT.button OR boxconveyor.jog.LDT.button OR panel.LDTJOG.LDT.button OR boxlongcutter.jog.LDT.button THEN
		jog := TRUE;
	ELSE
		jog := FALSE;
	END_IF
	IF 	boxunwinder.start.LDT.button OR boxwebbuffer.start.LDT.button OR boxcutting1.start.LDT.button
		(*OR boxlongcutter.start.LDT.button*) OR boxconveyor.start.LDT.button OR panel.LDTAutomatic.LDT.button THEN
		start := TRUE;
	ELSE
		start := FALSE;
	END_IF
	IF boxunwinder.stop.LDT.button AND  boxwebbuffer.stop.LDT.button AND  boxcutting1.stop.LDT.button
		(*AND  boxlongcutter.stop.LDT.button *)AND  boxconveyor.stop.LDT.button AND  panel.LDTStop.LDT.button THEN
		stop := TRUE;
	ELSE
		stop := FALSE;
	END_IF
	panel();
	boxunwinder(clk := clk);
	boxwebbuffer(clk := clk);
	boxcutting1(clk := clk);
	boxlongcutter(clk := clk);
	boxconveyor(clk := clk);
	clk();
END_FUNCTION_BLOCK
```

#### FB_SetCutOffset.st
```iecst
(********************************************************************
 * COPYRIGHT -- Microsoft
 ********************************************************************
 * Library: Bibliothek
 * Datei: SetCutOffset.st
 * Autor: okrebs
 * Erstellt: 23. Juli 2014
 ********************************************************************
 * Implementierung der Library Bibliothek
 ********************************************************************)

(* TODO: Bitte Kommentar hier einfügen *)
FUNCTION_BLOCK FB_SetCutOffset

	IF enable THEN

		IF UpdateRecipe THEN
			UpdateRecipe := FALSE;
			setvalueVisu := setvalueVisuRecipe/1000;
		END_IF

		Selectenable := TRUE;
		IF  step01 THEN
			step1 := FALSE;
			step10 := FALSE;
			step := 0.1;
			stepvisu := 0.1;
			Selectstep01 := TRUE;
			Selectstep1 := FALSE;
			Selectstep10 := FALSE;
		ELSIF step1 THEN
			step01 := FALSE;
			step10 := FALSE;
			step := 1;
			stepvisu := 1;
			Selectstep01 := FALSE;
			Selectstep1 := TRUE;
			Selectstep10 := FALSE;
		ELSIF step10 THEN
			step01 := FALSE;
			step1 := FALSE;
			step := 10;
			stepvisu := 10;
			Selectstep01 := FALSE;
			Selectstep1 := FALSE;
			Selectstep10 := TRUE;
		ELSE
			Selectstep01 := FALSE;
			Selectstep1 := FALSE;
			Selectstep10 := FALSE;
			step := 0;
		END_IF
		trigP(CLK := gearup );
		trigN(CLK := gearlow);
		IF trigP.Q AND setvalueVisu < limitvisupos - stepvisu THEN (*Stepper *)
			setvalueVisu := setvalueVisu + stepvisu;
		ELSIF trigN.Q AND setvalueVisu > limitvisuneg + stepvisu THEN
			setvalueVisu := setvalueVisu - stepvisu;
		END_IF

		IF setvalueVisu < -maxcorrection THEN
			setvalueVisu := -maxcorrection;
		ELSIF setvalueVisu > maxcorrection THEN
			setvalueVisu := maxcorrection;
		END_IF

//		setvalueVisu := LIMIT (-maxcorrection, REAL_TO_UDINT(setvalueVisu) ,maxcorrection);
	ELSE
		setvalueVisu := 0;

		Selectenable := FALSE;
	END_IF
	setOffset_o := REAL_TO_DINT(setvalueVisu * 1000);

END_FUNCTION_BLOCK
```

#### FB_SetGearRatio.st
```iecst
(********************************************************************
 * COPYRIGHT -- Microsoft
 ********************************************************************
 * Library: Bibliothek
 * Datei: FB_SetGearRatio.st
 * Autor: awalz
 * Erstellt: 2. Juli 2014
 ********************************************************************
 * Implementierung der Library Bibliothek
 ********************************************************************)

(* TODO: Bitte Kommentar hier einfügen *)
FUNCTION_BLOCK FB_SetGearRatio
	IF enable THEN
		Selectenable := TRUE;

		IF UpdateRecipe THEN
			UpdateRecipe := FALSE;
			setvalueVisu := setvalueVisuRecipe;
		END_IF
		offsetrecipe := setvalueVisuRecipe * 10;
		IF step1 THEN
			step10 := FALSE;
			step := 1;
			stepvisu :=0.1;
			Selectstep1 := TRUE;
			Selectstep10 := FALSE;
			Selectstep100 := FALSE;
		ELSIF step10 THEN
			step1 := FALSE;
			step := 10;
			stepvisu := 1;
			Selectstep1 := FALSE;
			Selectstep10 := TRUE;
			Selectstep100 := FALSE;
		ELSIF step100 THEN
			step1 := FALSE;
			stepvisu := 100;
			step := 100;
			Selectstep1 := FALSE;
			Selectstep10 := FALSE;
			Selectstep100 := TRUE;
		ELSE
			Selectstep1 := FALSE;
			Selectstep10 := FALSE;
			step := 0;
		END_IF
		trigP(CLK := gearup );
		trigN(CLK := gearlow);
		IF trigP.Q THEN (*Stepper *)
		 	ratio := ratio + step;
			setvalueVisu := setvalueVisu + stepvisu;
			Start_timer := TRUE;
			trigger := TRUE;
		ELSIF trigN.Q THEN
			ratio := ratio - step;
			setvalueVisu := setvalueVisu - stepvisu;
			Start_timer := TRUE;
			trigger := TRUE;
	 	END_IF
		(*ratioNumeratorOut:= LIMIT (800, ratio + REAL_TO_INT(offsetrecipe) ,1500) ;*)
		ratioNumeratorOut:= LIMIT (limitrationeg, ratio + REAL_TO_INT(offsetrecipe) ,limitratiopos);
		(*setvalueVisu := LIMIT (-20, setvalueVisu ,50);*)
		setvalueVisu := LIMIT (limitvisuneg, setvalueVisu ,limitvisupos);
		IF ratioNumeratorOut > ratioDenominator THEN
			ratio_inProcent_visu := (INT_TO_REAL(ratioNumeratorOut) - DINT_TO_REAL(ratioDenominator))/DINT_TO_REAL(ratioDenominator) *100;
		ELSE
			ratio_inProcent_visu := (INT_TO_REAL(ratioDenominator) - DINT_TO_REAL(ratioNumeratorOut))/DINT_TO_REAL(ratioDenominator) * -100;
		END_IF
		IF init THEN
			Start_timer := TRUE;
			trigger := TRUE;		// OKrebs 09.12.15
			init := FALSE;
		END_IF
		TP_01( IN:= Start_timer,PT:= T#1100ms);
		Start_timer := FALSE;
		IF NOT  TP_01.Q THEN
			trigger := FALSE;
		END_IF
	ELSE
		setvalueVisu := 0;
		ratioNumeratorOut := 1000;
		Selectenable := FALSE;
	END_IF
END_FUNCTION_BLOCK
```

#### FB_Alarme.st
```iecst
(********************************************************************
 * COPYRIGHT -- Microsoft
 ********************************************************************
 * Library: Bibliothek
 * Datei: FB_Alarme.st
 * Autor: okrebs
 * Erstellt: 1. August 2014
 ********************************************************************
 * Implementierung der Library Bibliothek
 ********************************************************************)

(* TODO: Bitte Kommentar hier einfügen *)
FUNCTION_BLOCK FB_Alarms

END_FUNCTION_BLOCK
```

#### FB_Liftcrtl.st
```iecst
(********************************************************************
 * COPYRIGHT -- Microsoft
 ********************************************************************
 * Library: Bibliothek
 * Datei: FB_Liftcrtl.st
 * Autor: awalz
 * Erstellt: 7. Oktober 2014
 ********************************************************************
 * Implementierung der Library Bibliothek
 ********************************************************************)

(* TODO: Bitte Kommentar hier einfügen *)
FUNCTION_BLOCK FB_Liftcrtl

buttomToggle(clk := clk);
	IF enable THEN
		IF buttomToggle.LDT.button AND NOT isdown THEN
			toUp_o := FALSE; (* wenn die Taste gedrück ist und unterer Ini noch nicht gekommen ist*)
			toDown_o := TRUE;
		ELSIF NOT isup AND NOT isdown AND NOT buttomToggle.LDT.button THEN (* soweit die Tatse los gelassen wird fährt die Zugstation nach oben*)
			toDown_o := FALSE;
			toUp_o := TRUE;
//		ELSIF  buttomToggle.LDT.button AND  isdown THEN (* soweit der untere Ini gekommen ist dauerhaft unten halten*)
//			toDown_o := FALSE;
//			toUp_o := TRUE;
		ELSIF buttomToggle.LDT.rtrig.Q AND isdown THEN (*einmalige Betätigung um die Zugstation hoch fahren lassen*)
			toDown_o :=FALSE;
			toUp_o := TRUE;
		END_IF
	END_IF
		IF init THEN
		toUp_o := TRUE;
		init := FALSE;
	END_IF

END_FUNCTION_BLOCK
```

#### FB_MachineSpeed.st
```iecst
(********************************************************************
 * COPYRIGHT -- Microsoft
 ********************************************************************
 * Library: Bibliothek
 * Datei: FB_MachineSpeed.st
 * Autor: awalz
 * Erstellt: 22. August 2014
 ********************************************************************
 * Implementierung der Library Bibliothek
 ********************************************************************)

(* TODO: Bitte Kommentar hier einfügen *)
FUNCTION_BLOCK FB_MachineSpeed
	lowPass.enable := TRUE;
	lowPass.x := INT_TO_REAL (dancepos);
	lowPass.t := 2;
	lowPass();
	lowPassSpeed.enable := TRUE;
	lowPassSpeed.x := INT_TO_REAL (ConveyerVelocity);
	lowPassSpeed.t := 2;
	lowPassSpeed();
//	lowPass.y_set := 0;
//	lowPass.set := TRUE;
//	rDancepos := INT_TO_REAL (dancepos) * SCALE_10V_TO_MM;
	rDancepos := lowPass.y * SCALE_10V_TO_MM;
	inc_to_volt := lowPassSpeed.y * SCALE_INC_TO_V;
	volt_to_speed := maxMainVelocity /10 * inc_to_volt;
	TP_01( IN:= Start_timer,PT:= T#600ms);
	Start_timer := TRUE;
	rtrig(CLK:= TP_01.Q); (*Die Position geht von oben 400 bis Tänzer unten 830 *)
	IF rDancepos > (setDancerpos + 50)  AND volt_to_speed > 0 THEN (*Tänzer ist unterhalb der Sollpos Maschine soll schneller laufen*)
		velocityOffset := (velocityOffset + 0.1(*velocityStep*));
		test := 1;
		Start_timer := FALSE; (*timer reset *)
	ELSIF rDancepos < (setDancerpos - 50) AND volt_to_speed > 0 THEN (*Tänzer ist oberhalb der Sollpos Maschine soll langsamer laufen*)
		velocityOffset := (velocityOffset - 0.1(*velocityStep*));
		test := 2;
		Start_timer := FALSE;
	ELSIF ( rDancepos  = highlimitDancerpos OR rDancepos < highlimitDancerpos )AND volt_to_speed > 0THEN
		velocityOffset := 0; (*oberer Anschlag*)
		test := 3;
		Start_timer := FALSE;
	ELSIF (rDancepos  = lowlimitDancerpos OR rDancepos >  lowlimitDancerpos ) AND volt_to_speed > 0THEN
		velocityOffset := 1;  (*unterer Anschlag*)
		test := 4;
		Start_timer := FALSE;
	ELSIF (setDancerpos + 50) > rDancepos AND rDancepos > (setDancerpos - 50) AND volt_to_speed > 0 THEN (* Fenster in dem die Maschine richtige geschwindigkeit hat*)
		velocityOffset := velocityOffset;
		test := 5;
		Start_timer := FALSE;
	ELSIF volt_to_speed = 0 OR volt_to_speed < 0 THEN
		velocityOffset := 0;
		test := 6;
	END_IF

	velocityramp.enable := TRUE;
	velocityramp.dy_down:= 0.1(* velocityStep*);
	velocityramp.dy_up	:= 0.1 (*velocityStep*);
	velocityramp.y_max := 1;
	velocityramp.y_min := -1;
	velocityramp.set := FALSE;
	velocityramp.x := velocityOffset;
	velocityramp();
	IF velocityramp.y <> 0 THEN
		tempvalue := floor(velocityramp.y* 10)/10;
	END_IF
	velocityOffset := LIMIT (-1, velocityOffset, 1);
//	IF reset THEN
//		setVelocity := 0;
//		(*actualVelocity := 0;*)
//		reset := FALSE;
//	END_IF
	IF reset THEN
		setVelocity := LIMIT (0, volt_to_speed, 21); (*setVelocity;*) (*+ velocityOffset;*) (* Offset damit der Tänzer in der Mitte bleibt*) // OKrebs // statt 11 -> 21
	ELSE
		setVelocity := LIMIT (0,( volt_to_speed + tempvalue), 21); // OKrebs // statt 11 -> 21
	END_IF

END_FUNCTION_BLOCK
```

#### FB_KeysWebbuffer.st
```iecst
(********************************************************************
 * COPYRIGHT -- Microsoft
 ********************************************************************
 * Library: Bibliothek
 * Datei: FB_KeysWebbuffer.st
 * Autor: awalz
 * Erstellt: 7. August 2014
 ********************************************************************
 * Implementierung der Library Bibliothek
 ********************************************************************)

(* TODO: Bitte Kommentar hier einfügen *)
FUNCTION_BLOCK FB_KeysWebbuffer
	up(clk:= clk);
	down(clk := clk);
	home(clk := clk);
	clk();
END_FUNCTION_BLOCK
```

#### FB_SwitchCabinet.st
```iecst
(********************************************************************
 * COPYRIGHT -- Microsoft
 ********************************************************************
 * Library: Bibliothek
 * Datei: FB_SwitchCabinet.st
 * Autor: awalz
 * Erstellt: 18. Juli 2014
 ********************************************************************
 * Implementierung der Library Bibliothek
 ********************************************************************)

(* TODO: Bitte Kommentar hier einfügen *)
FUNCTION_BLOCK FB_SwitchCabinet
EMCY_Buttons();
END_FUNCTION_BLOCK
```

#### Package Logical/Bibliothek/DATA - Neues leeres Paket

#### FB_WinderData.st
```iecst
(********************************************************************
 * COPYRIGHT -- Microsoft
 ********************************************************************
 * Library: Bibliothek
 * Datei: B_WinderData.st
 * Autor: Awalz
 * Erstellt: 14. Mai 2014
 ********************************************************************
 * Implementierung der Library Bibliothek
 ********************************************************************)

 (*<$Description$> TODO: Bitte Kommentar hier einzufügen </$Description$>*)
FUNCTION_BLOCK FB_WinderData
END_FUNCTION_BLOCK
```

#### FB_MASTERMODUL_DATA.st
```iecst
(********************************************************************
 * COPYRIGHT -- Microsoft
 ********************************************************************
 * Library: Bibliothek
 * Datei: FB_MASTERMODUL_DATA.st
 * Autor: Awalz
 * Erstellt: 14. Mai 2014
 ********************************************************************
 * Implementierung der Library Bibliothek
 ********************************************************************)

 (*<$Description$> TODO: Bitte Kommentar hier einzufügen </$Description$>*)
FUNCTION_BLOCK FB_MASTERMODUL_DATA
END_FUNCTION_BLOCK
```

#### FB_TENSIONMEASUREDATA.st
```iecst
(********************************************************************
 * COPYRIGHT -- Microsoft
 ********************************************************************
 * Library: Bibliothek
 * Datei: FB_TENSIONMEASUREDATA.st
 * Autor: Awalz
 * Erstellt: 12. Mai 2014
 ********************************************************************
 * Implementierung der Library Bibliothek
 ********************************************************************)

 (*<$Description$> TODO: Bitte Kommentar hier einzufügen </$Description$>*)
FUNCTION_BLOCK FB_TENSIONMEASUREDATA
END_FUNCTION_BLOCK
```

#### FB_CONVEYOR_DATA.st
```iecst
(********************************************************************
 * COPYRIGHT -- Microsoft
 ********************************************************************
 * Library: Bibliothek
 * Datei: FB_CONVEYOR_DATA.st
 * Autor: Awalz
 * Erstellt: 12. Mai 2014
 ********************************************************************
 * Implementierung der Library Bibliothek
 ********************************************************************)

 (*<$Description$> TODO: Bitte Kommentar hier einzufügen </$Description$>*)
FUNCTION_BLOCK FB_CONVEYOR_DATA
END_FUNCTION_BLOCK
```

#### FB_WinderMachData.st
```iecst
(********************************************************************
 * COPYRIGHT -- Microsoft
 ********************************************************************
 * Library: Bibliothek
 * Datei: FB_WinderMachData.st
 * Autor: Awalz
 * Erstellt: 14. Mai 2014
 ********************************************************************
 * Implementierung der Library Bibliothek
 ********************************************************************)

 (*<$Description$> TODO: Bitte Kommentar hier einzufügen </$Description$>*)
FUNCTION_BLOCK FB_WinderMachData
END_FUNCTION_BLOCK
```

#### FB_WinderRecipeData.st
```iecst
(********************************************************************
 * COPYRIGHT -- Microsoft
 ********************************************************************
 * Library: Bibliothek
 * Datei: FB_WinderRecipeData.st
 * Autor: Awalz
 * Erstellt: 14. Mai 2014
 ********************************************************************
 * Implementierung der Library Bibliothek
 ********************************************************************)

 (*<$Description$> TODO: Bitte Kommentar hier einzufügen </$Description$>*)
FUNCTION_BLOCK FB_WinderRecipeData
END_FUNCTION_BLOCK
```

#### FB_ScalingPerimeter.st
```iecst
(********************************************************************
 * COPYRIGHT -- Microsoft
 ********************************************************************
 * Library: Bibliothek
 * Datei: FB_FB_CuttingCalcScalingFactor.st
 * Autor: Awalz
 * Erstellt: 19. Mai 2014
 ********************************************************************
 * Implementierung der Library Bibliothek
 ********************************************************************)

 (*<$Description$> TODO: Bitte Kommentar hier einzufügen </$Description$>*)
FUNCTION_BLOCK FB_ScalingPerimeter
		IF (NumberToolSegments > 0) THEN
		Remainder	:= REAL_TO_DINT(floor(realperimeter) ) MOD USINT_TO_DINT(NumberToolSegments); (* Anzahl der Nutzen ohne den Restwert*)

		IF (Remainder > USINT_TO_DINT(NumberToolSegments / 2) ) THEN
			Remainder	:= Remainder - USINT_TO_DINT(NumberToolSegments);
		END_IF;

		Scaledperimeter	:= DINT_TO_UDINT(REAL_TO_DINT(floor(realperimeter) ) - Remainder);
		ToolSegmentPeriod	:= Scaledperimeter / NumberToolSegments;
	ELSE
		Scaledperimeter	:= 0;
		ToolSegmentPeriod	:= 0;
	END_IF;
END_FUNCTION_BLOCK
```

#### FB_CUTTINGUNIT_STATUS.st
```iecst
(********************************************************************
 * COPYRIGHT -- Microsoft
 ********************************************************************
 * Library: Bibliothek
 * Datei: FB_CUTTINGUNIT_STATUS.st
 * Autor: Awalz
 * Erstellt: 20. Mai 2014
 ********************************************************************
 * Implementierung der Library Bibliothek
 ********************************************************************)

 (*<$Description$> TODO: Bitte Kommentar hier einzufügen </$Description$>*)
FUNCTION_BLOCK FB_CUTTINGUNIT_STATUS

	IF dataOk AND mode.value = recipeMode THEN
		IF mode.value = CONST.CUTTINGUNIT.MODEs.DISABLE THEN  (* wenn disabled alles bereit melden*)
			ready := TRUE;
			tmpCalibrated := TRUE;
		ELSE
			ready := isCoupled AND extReady;
			tmpCalibrated := isCalibrated;
		END_IF
	ELSE
		ready := FALSE;
		tmpCalibrated := isCalibrated;
	END_IF
	IF axisState.ContinuousMotion THEN
		AxisState_status := 'ContinuousMotion';
	ELSIF axisState.Disabled THEN
		AxisState_status := 'Disabled';
	ELSIF axisState.DiscreteMotion THEN
		AxisState_status := 'DiscreteMotion';
	ELSIF axisState.Error THEN
		AxisState_status := 'Error';
	ELSIF axisState.Errorstop THEN
		AxisState_status := 'Errorstop';
	ELSIF axisState.StandStill THEN
		AxisState_status := 'StandStill';
	ELSIF axisState.Stopping THEN
		AxisState_status := 'Stopping';
	ELSIF axisState.SynchronizedMotion THEN
		AxisState_status := 'SynchronizedMotion';
	END_IF
END_FUNCTION_BLOCK
```

#### FB_CROSSCUTPAR.st
```iecst
(********************************************************************
 * COPYRIGHT -- Microsoft
 ********************************************************************
 * Library: Bibliothek
 * Datei: FB_CROSSCUTPAR.st
 * Autor: awalz
 * Erstellt: 8. Juli 2014
 ********************************************************************
 * Implementierung der Library Bibliothek
 ********************************************************************)

(* TODO: Bitte Kommentar hier einfügen *)
FUNCTION_BLOCK FB_CROSSCUTPAR
END_FUNCTION_BLOCK
```

#### FB_PACKBELT_DATA.st
```iecst
(********************************************************************
 * COPYRIGHT -- Microsoft
 ********************************************************************
 * Library: Bibliothek
 * Datei: FB_PACKBELT_DATA.st
 * Autor: okrebs
 * Erstellt: 10. Januar 2017
 ********************************************************************
 * Implementierung der Library Bibliothek
 ********************************************************************)

(* TODO: Bitte Kommentar hier einfügen *)
FUNCTION_BLOCK FB_PACKBELT_DATA
END_FUNCTION_BLOCK
```

#### Package Logical/Bibliothek/Axis - Paket

#### FB_AxisCtrl.st
```iecst
(********************************************************************
 * COPYRIGHT -- Microsoft
 ********************************************************************
 * Library: Bibliothek
 * Datei: FB_AxisCtrl.st
 * Autor: awalz
 * Erstellt: 23. Juli 2014
 ********************************************************************
 * Implementierung der Library Bibliothek
 ********************************************************************)

(* TODO: Bitte Kommentar hier einfügen *)
FUNCTION_BLOCK FB_AxisCtrl

(***************************************************************
        Control Sequence
***************************************************************)
(* status information is read before the step sequencer to attain a shorter reaction time *)
(************************ MC_READSTATUS *************************)
	MC_ReadStatus_0.Enable :=  NOT MC_ReadStatus_0.Error;
	MC_ReadStatus_0.Axis := AxisREF;
	MC_ReadStatus_0();
	BasicControl.AxisState.Disabled             := MC_ReadStatus_0.Disabled;
	BasicControl.AxisState.StandStill           := MC_ReadStatus_0.StandStill;
	BasicControl.AxisState.Stopping             := MC_ReadStatus_0.Stopping;
	BasicControl.AxisState.Homing               := MC_ReadStatus_0.Homing;
	BasicControl.AxisState.DiscreteMotion       := MC_ReadStatus_0.DiscreteMotion;
	BasicControl.AxisState.ContinuousMotion     := MC_ReadStatus_0.ContinuousMotion;
	BasicControl.AxisState.SynchronizedMotion   := MC_ReadStatus_0.SynchronizedMotion;
	BasicControl.AxisState.ErrorStop            := MC_ReadStatus_0.Errorstop;

	(********************MC_BR_READDRIVESTATUS***********************)
	MC_BR_ReadDriveStatus_0.Enable := NOT(MC_BR_ReadDriveStatus_0.Error);
	MC_BR_ReadDriveStatus_0.Axis := AxisREF;
	MC_BR_ReadDriveStatus_0.AdrDriveStatus := ADR(BasicControl.Status.DriveStatus);
	MC_BR_ReadDriveStatus_0();

	(******************** MC_READACTUALPOSITION *********************)
	MC_ReadActualPosition_0.Enable := (NOT(MC_ReadActualPosition_0.Error));
	MC_ReadActualPosition_0.Axis := AxisREF;
	MC_ReadActualPosition_0();
	IF(MC_ReadActualPosition_0.Valid = TRUE)THEN
		BasicControl.Status.ActPosition := MC_ReadActualPosition_0.Position;
	END_IF

	(******************** MC_READACTUALVELOCITY *********************)
	MC_ReadActualVelocity_0.Enable := (NOT(MC_ReadActualVelocity_0.Error));
	MC_ReadActualVelocity_0.Axis := AxisREF;
	MC_ReadActualVelocity_0();
	IF(MC_ReadActualVelocity_0.Valid = TRUE)THEN
		BasicControl.Status.ActVelocity := MC_ReadActualVelocity_0.Velocity;
	END_IF
	(*********************+*Parameter schreiben**********************)
	MC_MoveVelocity_0.Acceleration  := ruck;
	MC_MoveVelocity_0.Deceleration  := ruck;
	MC_ReadStatus_0();
	(************************ MC_READAXISERROR **********************)
	MC_ReadAxisError_0.Enable := NOT(MC_ReadAxisError_0.Error);
	MC_ReadAxisError_0.Axis := AxisREF;
	MC_ReadAxisError_0.DataAddress := ADR(BasicControl.Status.ErrorText);
	MC_ReadAxisError_0.DataLength := SIZEOF(BasicControl.Status.ErrorText);
	MC_ReadAxisError_0.DataObjectName := 'acp10etxde';
	MC_ReadAxisError_0();
	(* central monitoring OF stop command attains a shorter reaction TIME in CASE OF emergency stop *)
	(******************CHECK FOR STOP COMMAND************************)
	(*IF (BasicControl.Command.Stop = TRUE) THEN*)
//	IF cmd = CONST.AXIS.STOP THEN //12.03.15
//		busy := TRUE;
//		IF ((AxisStep >= STATE_READY) AND (AxisStep < STATE_ERROR)) THEN
//			(* reset all FB execute inputs we use *)
//			MC_Home_0.Execute := 0;
//			MC_Stop_0.Execute := 0;
//			MC_MoveAbsolute_0.Execute := 0;
//			MC_MoveAdditive_0.Execute := 0;
//			MC_MoveVelocity_0.Execute := 0;
//			MC_ReadAxisError_0.Acknowledge := 0;
//			MC_Reset_0.Execute := 0;
//
//			(* reset user commands *)
//			BasicControl.Command.Stop := 0;
//			BasicControl.Command.Home := 0;
//			BasicControl.Command.MoveJogPos := 0;
//			BasicControl.Command.MoveJogNeg := 0;
//			BasicControl.Command.MoveVelocity := 0;
//			BasicControl.Command.MoveAbsolute := 0;
//			BasicControl.Command.MoveAdditive := 0;
//			MC_Stop_0( Execute := TRUE, Deceleration := verzoegerung);
//			AxisStep := STATE_STOP;
//		END_IF
//	END_IF
//
////////////////////////////////////////////////////////////////////////////
//(*	IF AxisHandle[tempIndex].AxisState.Stopping THEN
//	    IF (AxisHandle[tempIndex].Status.ActVelocity = 0.0) THEN
//			AxisIf.Status.isMoving 						:= FALSE;
//			AllDrives.Status.stopActive					:= FALSE;
//		ELSE
//			AxisIf.Status.isMoving 						:= TRUE;
//		END_IF
//	ELSIF (NOT ( AxisHandle[tempIndex].AxisState.DiscreteMotion OR
//	             AxisHandle[tempIndex].AxisState.ContinuousMotion)) THEN
//		AxisIf.Status.isMoving 							:= FALSE;
//		AllDrives.Status.stopActive						:= FALSE;
//	ELSE
//		AxisIf.Status.isMoving 							:= TRUE;
//	END_IF*)
//////////////////////////////////////////////////////////////////////////////
//	(**************** CHECK FOR GENERAL AXIS ERROR ******************)
//(*	IF ((MC_ReadAxisError_0.AxisErrorID <> 0) AND (MC_ReadAxisError_0.Valid)) THEN
//		AxisStep := STATE_ERROR_AXIS;
//		(***************** CHECK IF POWER SHOULD BE OFF *******************)
//(*	ELSIF ((NOT BasicControl.Command.Power) AND (MC_ReadAxisError_0.Valid)) THEN
//		IF ((MC_ReadStatus_0.Errorstop) AND (MC_ReadStatus_0.Valid )) THEN
//			AxisStep := STATE_ERROR_RESET;
//		ELSE
//			AxisStep := STATE_WAIT;
//		END_IF
//	END_IF*)

	CASE AxisStep OF

//		******************* WAIT ************************
		STATE_WAIT:  (* STATE: Wait *)
			AxisStep := STATE_QUIT;
//			(*IF (BasicControl.Command.Power = TRUE) THEN*)
//			IF cmd = CONST.AXIS.POWER_ON THEN
//				cmdtmp := cmd;
//				AxisStep := STATE_POWER_ON;
//			ELSIF cmd = CONST.AXIS.VAXIS_ON THEN
//				cmdtmp := cmd;
//				AxisStep := STATE_VAXIS_ON;
//			ELSIF cmd = CONST.AXIS.POWER_OFF THEN
//				cmdtmp := cmd;
//				AxisStep := STATE_POWER_OFF;
//			ELSE
//				MC_Power_0.Enable := FALSE;
//			END_IF
//
//			(* reset all FB execute inputs we use *)
//			MC_Home_0.Execute := FALSE;
//			MC_Stop_0.Execute := FALSE;
//			MC_MoveAbsolute_0.Execute := FALSE;
//			MC_MoveAdditive_0.Execute := FALSE;
//			MC_MoveVelocity_0.Execute := FALSE;
//			MC_ReadAxisError_0.Acknowledge := FALSE;
//			MC_Reset_0.Execute := FALSE;
//			(* reset user commands *)
//			BasicControl.Command.Stop := FALSE;
//			BasicControl.Command.Home := FALSE;
//			BasicControl.Command.MoveJogPos := FALSE;
//			BasicControl.Command.MoveJogNeg := FALSE;
//			BasicControl.Command.MoveVelocity := FALSE;
//			BasicControl.Command.MoveAbsolute := FALSE;
//			BasicControl.Command.MoveAdditive := FALSE;
//
//			BasicControl.Status.ErrorID := 0;
//		(********************Virtuelle Achse einschalten****)
		STATE_VAXIS_ON:

			IF MC_BR_ReadDriveStatus_0.Valid THEN
				cmdtmp := cmd;
				AxisStep := STATE_QUIT;
			END_IF
		(******************** POWER ON **********************)
		STATE_POWER_ON:  (* STATE: Power on *)
			(*MC_Power_0.Enable := TRUE;*)
			IF BasicControl.Status.DriveStatus.ControllerReady AND	cmd = CONST.AXIS.POWER_ON
				AND NOT MC_Power_0.Status AND NOT MC_Power_0.Error THEN
				MC_Power_0.Enable := TRUE; (*erster Anlauf*)
					cmdtmp := cmd;
			ELSIF MC_Power_0.Error AND cmdtmp = cmd THEN
					MC_Power_0.Enable := FALSE ;(* if a power error occured go to error state *)
					cmd := CONST.AXIS.RESET;
					AxisStep := STATE_ERROR_RESET;
			ELSIF 	MC_Power_0.Status AND NOT MC_Power_0.Error THEN
					cmdtmp := cmd;
					AxisStep := STATE_QUIT;
		(*	ELSIF MC_Power_0.Error AND cmdtmp <> cmd THEN
					BasicControl.Status.ErrorID := MC_Power_0.ErrorID;
					AxisStep := STATE_ERROR;*)
			ELSIF MC_ReadStatus_0.Errorstop THEN (*24.07.14*)
					BasicControl.Status.ErrorID := MC_Power_0.ErrorID;
					cmdtmp := cmd;
					AxisStep := STATE_ERROR;
			END_IF
		(******************** POWER OFF **********************)
		STATE_POWER_OFF:  (* STATE: Power on *)
			MC_Power_0.Enable := FALSE;
			IF NOT MC_Power_0.Status THEN
				cmdtmp := cmd;
				(*AxisStep := STATE_READY;*)
				AxisStep := STATE_QUIT;
			END_IF
			(* if a power error occured go to error state *)
			IF MC_Power_0.Error  THEN
				BasicControl.Status.ErrorID := MC_Power_0.ErrorID;
				AxisStep := STATE_ERROR;
			END_IF
		(******************** READY **********************)
		STATE_READY:  (* STATE: Waiting for commands *)
			IF cmd <> CONST.AXIS.NOACTION THEN
					busy := TRUE;
					(*cmdtmp:= cmd; *)//13.03.15
					IF cmd = CONST.AXIS.RESET THEN
						AxisStep := STATE_ERROR_RESET;
					ELSIF cmd = CONST.AXIS.STOP THEN
						MC_Stop_0( Execute := TRUE, Deceleration := verzoegerung);
						AxisStep := STATE_STOP;
					ELSIF cmd = CONST.AXIS.JOG_NEG THEN
						MC_MoveVelocity_0(Execute := TRUE, Velocity := 16666*velocity, Acceleration := BasicControl.Parameter.Acceleration,
										Deceleration  := BasicControl.Parameter.Deceleration, Direction := mcNEGATIVE_DIR);
						AxisStep := STATE_JOG_NEGATIVE;
					ELSIF cmd = CONST.AXIS.JOG_POS THEN
						MC_MoveVelocity_0(Execute := TRUE, Velocity := 16666*velocity, Acceleration := BasicControl.Parameter.Acceleration,
										Deceleration  := BasicControl.Parameter.Deceleration,Direction := mcPOSITIVE_DIR);
						AxisStep := STATE_JOG_POSITIVE;
					ELSIF cmd = CONST.AXIS.SETPOS THEN
						MC_MoveAbsolute_0(Execute := TRUE, Position := position, Velocity := 16666*velocity, Acceleration := BasicControl.Parameter.Acceleration,
										Deceleration  := BasicControl.Parameter.Deceleration, Direction := mcPOSITIVE_DIR);
						AxisStep := STATE_MOVE_ABSOLUTE;
					ELSIF  cmd = CONST.AXIS.CALIBR THEN
						(*Achse referenzieren*)
						AxisStep := STATE_HOME;
					ELSIF cmd = CONST.AXIS.MOVE_VELOCITY THEN
//							MC_MoveVelocity_0.Acceleration  := BasicControl.Parameter.Acceleration;
//							MC_MoveVelocity_0.Deceleration  := BasicControl.Parameter.Deceleration;
							MC_MoveVelocity_0(Execute := TRUE, Velocity := 16666*velocity, Acceleration := BasicControl.Parameter.Acceleration,
												Deceleration  := BasicControl.Parameter.Deceleration,	Direction := mcPOSITIVE_DIR);
						AxisStep := STATE_MOVE_VELOCITY;
					ELSIF   cmd = CONST.AXIS.POWER_OFF THEN
						AxisStep := STATE_POWER_OFF;
					ELSIF   cmd = CONST.AXIS.POWER_ON THEN
						AxisStep := STATE_POWER_ON;
					END_IF
			ELSE
				busy := FALSE;
			END_IF
		(******************** HOME **********************)
		STATE_HOME:  (* STATE: start homing process *)
			MC_Home_0.Position := BasicControl.Parameter.HomePosition;
			MC_Home_0.HomingMode := BasicControl.Parameter.HomeMode;
			MC_Home_0.HomingMode := mcHOME_SWITCH_GATE;
			MC_Home_0.Execute := TRUE;
			IF MC_Home_0.Done AND cmd = CONST.AXIS.CALIBR THEN
				MC_Home_0.Execute := FALSE;
				BasicControl.AxisState.Homed := TRUE;
				cmdtmp := cmd;
				AxisStep := STATE_QUIT;
			ELSIF cmd <> CONST.AXIS.CALIBR THEN
				MC_Home_0.Execute := FALSE;
				MC_Stop_0( Execute := TRUE, Deceleration := verzoegerung);
				AxisStep := STATE_STOP;
			END_IF

			(* if a homing error occured go to error state *)
			IF MC_Home_0.Error  OR MC_ReadStatus_0.Errorstop THEN
				MC_Home_0.Execute := FALSE;
				BasicControl.Status.ErrorID := MC_Home_0.ErrorID;
				AxisStep := STATE_ERROR;
			END_IF

		(***********************HALT_MOVEMENT***************************)
		STATE_HALT:   (* STATE: Halt movement *)
			MC_Halt_0.Deceleration := BasicControl.Parameter.Deceleration;
			MC_Halt_0.Execute := TRUE;
			IF MC_Halt_0.Done THEN
				MC_Halt_0.Execute := FALSE;
				cmdtmp := cmd;
				AxisStep := STATE_QUIT;
			ELSIF cmd = CONST.AXIS.STOP THEN
				MC_Halt_0.Execute := FALSE;
				MC_Stop_0( Execute := TRUE, Deceleration := verzoegerung);
				AxisStep := STATE_STOP;
			END_IF
			(* check if error occured *)
			IF MC_Halt_0.Error OR  MC_ReadStatus_0.Errorstop THEN
				BasicControl.Status.ErrorID := MC_Halt_0.ErrorID;
				MC_Halt_0.Execute := FALSE;
				AxisStep := STATE_ERROR;
			END_IF

		(*********************** STOP MOVEMENT *************************)
		STATE_STOP:  (* STATE: Stop movement *)
//			MC_Stop_0.Deceleration := BasicControl.Parameter.Deceleration;
//			MC_Stop_0.Execute := TRUE;
			(* if axis is stopped go to ready state *)
			IF MC_Stop_0.Done  OR MC_ReadStatus_0.StandStill THEN
				MC_Stop_0.Execute := FALSE;
				cmdtmp := cmd;
				AxisStep := STATE_QUIT;
			ELSIF MC_ReadStatus_0.Disabled THEN
				MC_Stop_0.Execute := FALSE;
				cmdtmp := cmd;
				AxisStep := STATE_QUIT;
			END_IF
			(* check if error occured *)
			IF MC_Stop_0.Error OR MC_ReadStatus_0.Errorstop THEN
				BasicControl.Status.ErrorID := MC_Stop_0.ErrorID;
				MC_Stop_0.Execute := FALSE;
				AxisStep := STATE_ERROR;
			END_IF

		(******************** START JOG MOVEMENT POSITVE **********************)
		STATE_JOG_POSITIVE:  (* STATE: Start jog movement in positive direction *)
			IF cmd <> CONST.AXIS.JOG_POS AND cmd <> CONST.AXIS.STOP THEN
				cmdtmp := cmd;
				MC_MoveVelocity_0.Execute := FALSE;
				AxisStep := STATE_HALT;
			ELSIF cmd = CONST.AXIS.STOP THEN
				MC_MoveVelocity_0.Execute := FALSE;
				MC_Stop_0( Execute := TRUE, Deceleration := verzoegerung);
				AxisStep := STATE_STOP;
			END_IF
			(* check if error occured *)
			IF MC_MoveVelocity_0.Error OR MC_ReadStatus_0.Errorstop  THEN
				BasicControl.Status.ErrorID := MC_MoveVelocity_0.ErrorID;
				MC_MoveVelocity_0.Execute := FALSE;
				AxisStep := STATE_ERROR;
			END_IF

		(******************** START JOG MOVEMENT NEGATIVE **********************)
		STATE_JOG_NEGATIVE:  (* STATE: Start jog movement in negative direction *)
			IF cmd <> CONST.AXIS.JOG_NEG AND cmd <> CONST.AXIS.STOP  THEN
				MC_MoveVelocity_0.Execute := FALSE;
				cmdtmp := cmd;
				AxisStep := STATE_HALT;
			ELSIF cmd = CONST.AXIS.STOP THEN
				MC_MoveVelocity_0.Execute := FALSE;
				MC_Stop_0( Execute := TRUE, Deceleration := verzoegerung);
				AxisStep := STATE_STOP;
			END_IF
			(* check if error occured *)
			IF MC_MoveVelocity_0.Error OR MC_ReadStatus_0.Errorstop  THEN
				BasicControl.Status.ErrorID := MC_MoveVelocity_0.ErrorID;
				MC_MoveVelocity_0.Execute := FALSE;
				AxisStep := STATE_ERROR;
			END_IF

		(******************** START ABSOLUTE MOVEMENT **********************)
		STATE_MOVE_ABSOLUTE:  (* STATE: Start absolute movement *)
			(* check if commanded position is reached *)
			IF cmd <> CONST.AXIS.SETPOS AND cmd <> CONST.AXIS.STOP THEN
				MC_MoveAbsolute_0.Execute := FALSE;
				cmdtmp := cmd;
				AxisStep := STATE_HALT;
			ELSIF MC_MoveAbsolute_0.Done  THEN
				MC_MoveAbsolute_0.Execute := FALSE;
				cmdtmp := cmd;
				AxisStep := STATE_QUIT;
			ELSIF cmd = CONST.AXIS.STOP THEN
				MC_MoveAbsolute_0.Execute := FALSE;
				MC_Stop_0( Execute := TRUE, Deceleration := verzoegerung);
				AxisStep := STATE_STOP;
			END_IF
			(* check if error occured *)
			IF MC_MoveAbsolute_0.Error OR MC_ReadStatus_0.Errorstop THEN
				BasicControl.Status.ErrorID := MC_MoveAbsolute_0.ErrorID;
				MC_MoveAbsolute_0.Execute := TRUE;
				AxisStep := STATE_ERROR;
			END_IF

		(******************** START ADDITIVE MOVEMENT **********************)
		STATE_MOVE_ADDITIVE:  (* STATE: Start additive movement *)
			(* check if commanded distance is reached *)
			IF cmd <> CONST.AXIS.SETPOS AND cmd <> CONST.AXIS.STOP THEN
				MC_MoveAdditive_0.Execute := FALSE;
				cmdtmp := cmd;
				AxisStep := STATE_HALT;
				AxisStep := STATE_HALT;
			ELSIF MC_MoveAdditive_0.Done THEN
				MC_MoveAdditive_0.Execute := FALSE;
				cmdtmp := cmd;
				AxisStep := STATE_QUIT;
			ELSIF cmd = CONST.AXIS.STOP THEN
				MC_MoveAdditive_0.Execute := FALSE;
				MC_Stop_0( Execute := TRUE, Deceleration := verzoegerung);
				AxisStep := STATE_STOP;
			END_IF
			(* check if error occured *)
			IF MC_MoveAdditive_0.Error OR  MC_ReadStatus_0.Errorstop THEN
				BasicControl.Status.ErrorID := MC_MoveAdditive_0.ErrorID;
				MC_MoveAdditive_0.Execute := FALSE;
				AxisStep := STATE_ERROR;
			END_IF

		(******************** START VELOCITY MOVEMENT **********************)
		STATE_MOVE_VELOCITY:  (* STATE: Start velocity movement *)
			IF cmd <>  CONST.AXIS.MOVE_VELOCITY AND  cmd <> CONST.AXIS.STOP THEN
				MC_MoveVelocity_0.Execute := FALSE;
				cmdtmp := cmd;
				AxisStep := STATE_HALT;
			ELSIF MC_MoveVelocity_0.InVelocity THEN
				MC_MoveVelocity_0.Execute := FALSE;
				cmdtmp := cmd;
				AxisStep := STATE_QUIT;
			ELSIF cmd = CONST.AXIS.STOP THEN
				MC_MoveVelocity_0.Execute := FALSE;
				MC_Stop_0( Execute := TRUE, Deceleration := verzoegerung);
				AxisStep := STATE_STOP;
			END_IF
			(* check if error occured *)
			IF MC_MoveVelocity_0.Error OR MC_ReadStatus_0.Errorstop  THEN
				BasicControl.Status.ErrorID := MC_MoveVelocity_0.ErrorID;
				MC_MoveVelocity_0.Execute := FALSE;
				AxisStep := STATE_ERROR;
			END_IF

		(******************** FB-ERROR OCCURED *************************)
		STATE_ERROR:  (* STATE: Error *)
			(* check if FB indicates an axis error *)
			IF (MC_ReadAxisError_0.AxisErrorCount<>0) THEN
				AxisStep := STATE_ERROR_AXIS;
			ELSE
				IF (BasicControl.Command.ErrorAcknowledge = TRUE) THEN
					BasicControl.Command.ErrorAcknowledge := FALSE;
					BasicControl.Status.ErrorID := 0;
					(* reset axis if it is in axis state ErrorStop *)
					IF MC_ReadStatus_0.Errorstop AND MC_ReadStatus_0.Valid  THEN
						AxisStep := STATE_ERROR_RESET;
					ELSE
						(*AxisStep := STATE_WAIT;*)
							cmdtmp := cmd;
						AxisStep := STATE_QUIT;
					END_IF
				END_IF
			END_IF

		(******************** AXIS-ERROR OCCURED *************************)
		STATE_ERROR_AXIS:  (* STATE: Axis Error *)
			IF (MC_ReadAxisError_0.Valid) THEN
			err.set := TRUE;
			err.text := MC_ReadAxisError_0.DataObjectName;
			err.id :=  UINT_TO_DINT  (MC_ReadAxisError_0.AxisErrorID) ;
				IF (MC_ReadAxisError_0.AxisErrorID <> 0) THEN
					BasicControl.Status.ErrorID := MC_ReadAxisError_0.AxisErrorID;
				END_IF
				MC_ReadAxisError_0.Acknowledge := FALSE;
			(*	IF (BasicControl.Command.ErrorAcknowledge) THEN
					BasicControl.Command.ErrorAcknowledge := FALSE;
					(* acknowledge axis error *)
				IF cmd = CONST.AXIS.RESET THEN
					IF (MC_ReadAxisError_0.AxisErrorID <> 0) THEN
						MC_ReadAxisError_0.Acknowledge := TRUE;
						AxisStep := STATE_ERROR_RESET;
					END_IF
				END_IF
				IF (MC_ReadAxisError_0.AxisErrorCount = 0) THEN
					(* reset axis if it is in axis state ErrorStop *)
					BasicControl.Status.ErrorID := 0;
					IF ((MC_ReadStatus_0.Errorstop ) AND (MC_ReadStatus_0.Valid)) THEN
						AxisStep := STATE_ERROR_RESET;
					ELSE
						(*AxisStep := STATE_WAIT;*)
						cmdtmp := cmd;
						AxisStep := STATE_QUIT;
					END_IF
				ELSIF NOT MC_ReadAxisError_0.Error THEN
							cmdtmp := cmd;
							AxisStep := STATE_QUIT;
				END_IF
			ELSE
				AxisStep := STATE_WAIT; (* kein Fehler liegt vor*)
			END_IF

		(******************** RESET DONE *************************)
		STATE_ERROR_RESET:  (* STATE: Wait for reset done *)
			MC_Reset_0.Execute := TRUE;
			(* reset MC_Power.Enable if this FB is in Error*)
			IF (MC_Power_0.Error) THEN
				MC_Power_0.Enable := FALSE;
			END_IF
			IF(MC_Reset_0.Done)THEN
				MC_Reset_0.Execute := FALSE;
				cmdtmp := cmd;
				AxisStep := STATE_QUIT;
			ELSIF(MC_Reset_0.Error) THEN
				MC_Reset_0.Execute := FALSE;
				AxisStep := STATE_ERROR;
			END_IF
			(******************** SEQUENCE END *************************)
		STATE_QUIT:
			busy := FALSE;
			IF cmd = cmdtmp THEN
				busy := FALSE;
				cmd := CONST.AXIS.NOACTION;
				AxisStep := STATE_READY;
			ELSIF cmd <> CONST.AXIS.NOACTION THEN
				busy := FALSE;
				AxisStep := STATE_READY;
			END_IF

	END_CASE

(***************************************************************
        Function Block Calls
***************************************************************)

(************************** MC_POWER ****************************)
	MC_Power_0.Axis := AxisREF;  (* pointer to axis *)
	MC_Power_0();

	(************************** MC_HOME *****************************)
	MC_Home_0.Axis := AxisREF;
	MC_Home_0();

	(********************** MC_MOVEABSOLUTE *************************)
	MC_MoveAbsolute_0.Acceleration := BasicControl.Parameter.Acceleration;
	MC_MoveAbsolute_0.Deceleration := BasicControl.Parameter.Deceleration;
	MC_MoveAbsolute_0.Axis := AxisREF;
	MC_MoveAbsolute_0();

	(********************** MC_MOVEADDITIVE *************************)
	MC_MoveAdditive_0.Acceleration := BasicControl.Parameter.Acceleration;
	MC_MoveAdditive_0.Deceleration := BasicControl.Parameter.Deceleration;
	MC_MoveAdditive_0.Axis := AxisREF;
	MC_MoveAdditive_0();

	(********************** MC_MOVEVELOCITY *************************)
	MC_MoveVelocity_0.Acceleration  := BasicControl.Parameter.Acceleration;
	MC_MoveVelocity_0.Deceleration  := BasicControl.Parameter.Deceleration;
	MC_MoveVelocity_0.Axis := AxisREF;
	MC_MoveVelocity_0();

	(************************** MC_STOP *****************************)
	MC_Stop_0.Axis := AxisREF;
	MC_Stop_0();

	(***************************MC_HALT******************************)
	MC_Halt_0.Axis := AxisREF;
	MC_Halt_0();

	(************************** MC_RESET ****************************)
	MC_Reset_0.Axis := AxisREF;
	MC_Reset_0();

END_FUNCTION_BLOCK
```
